FUNCTION_BLOCK FB_Power_lever
VAR_INPUT
	Forward:BOOL; (*Lever notch 1 forward*)
	Reverse:BOOL; (*Lever notch 1 reverse*)
	Pot:INT; (*Analogue value from lever potentiometer*)
	Button:BOOL;
	Neutral:BOOL; 
	Use_neutral:BOOL;
	Fully_fwd_val:INT; (*Value of analogue input when lever is fully forward*)
	Fully_rev_val:INT; (*Value of analogue input when lever is fully reverse*)
	Zero_deadband:INT; (*Lever zero position deadband on a scale of 0 to 10 000 i.e. a value of 100 gives a 1% deadband in each direction*)
	Full_lever_deadband:INT; (*Lever fully forward or reverse deadband on a scale of 0 to 10 000 i.e. a value of 100 gives a 1% deadband*)
	Notch_position:INT; (*Lever value (-10 000 to 10 000, no deadbands) at which forward and reverse notches change state*)
	Allowed_notch_variation:INT; (*Allowed variation in notch position*)
	Pos_out_of_range_val:INT; (*If the analogue Pot value exceeds this threshold, a fault will be generated.*)
	Neg_out_of_range_val:INT; (*If the analogue Pot value is less than this threshold, a fault will be generated.*)
END_VAR
VAR_OUTPUT
	Power_lever_data:dut_Power_lever;
	Raw:INT; (*Linear scaled lever value with no deadbands applied. -10 000 = fully reverse. +10 000 = fully forward.*)
	Linear:INT; (*Linear scaled lever value with deadbands applied. -10 000 = fully reverse. +10 000 = fully forward.*)
	Cubic:INT; (*Cubic scaling applied to lever value with deadbands applied. -10 000 = fully reverse. +10 000 = fully forward.*)
	cs_Forward_and_reverse:BOOL; (*Forward and reverse inputs both energised.*)
	cs_Pot_fwd_no_notch:BOOL; (*Pot shows that lever is forward but the forward notch is not activated*)
	cs_Pot_rev_no_notch:BOOL; (*Pot shows that lever is reverse but the reverse notch is not activated*)
	cs_Fwd_notch_not_pot:BOOL; (*Reverse notch is activated but the pot does not show that the lever is past the reverse notch*)
	cs_Rev_notch_not_pot:BOOL; (*Forward notch is activated but the pot does not show that the lever is past the forward notch*)
	cs_Out_of_range_pos:BOOL; (*The Pot value is out of range in the positive direction*)
	cs_Out_of_range_neg:BOOL; (*The Pot value is out of range in the negative direction*)
	hmi_data:dut_hmi_Power_lever; (*HMI status bits as well as Raw, Linear and Cubic values*)
END_VAR
VAR
	Linear_abs: INT;
	hmi_Word:WORD;
	TON_0: TON;
	TON_2: TON;
	TON_1: TON;
	TON_3: TON;
	Lever_scaling: Lever_scaling;
	Power_lever_data_m: Power_lever_data;
	Power_lever_faults: Power_lever_faults;
	BIT_TO_WORD_V0_0: FB_BIT_TO_WORD_V0;
END_VAR

Lever_scaling();
Power_lever_data_m();
Power_lever_faults();

METHOD Lever_scaling
VAR_INPUT
END_VAR
VAR_INST // added by the converter: edge detectors and wires of the graphical bodies
    _w1, _w2, _w3, _w4, _w5, _w6, _w8 : ANY;
    _w7 : REAL;
END_VAR
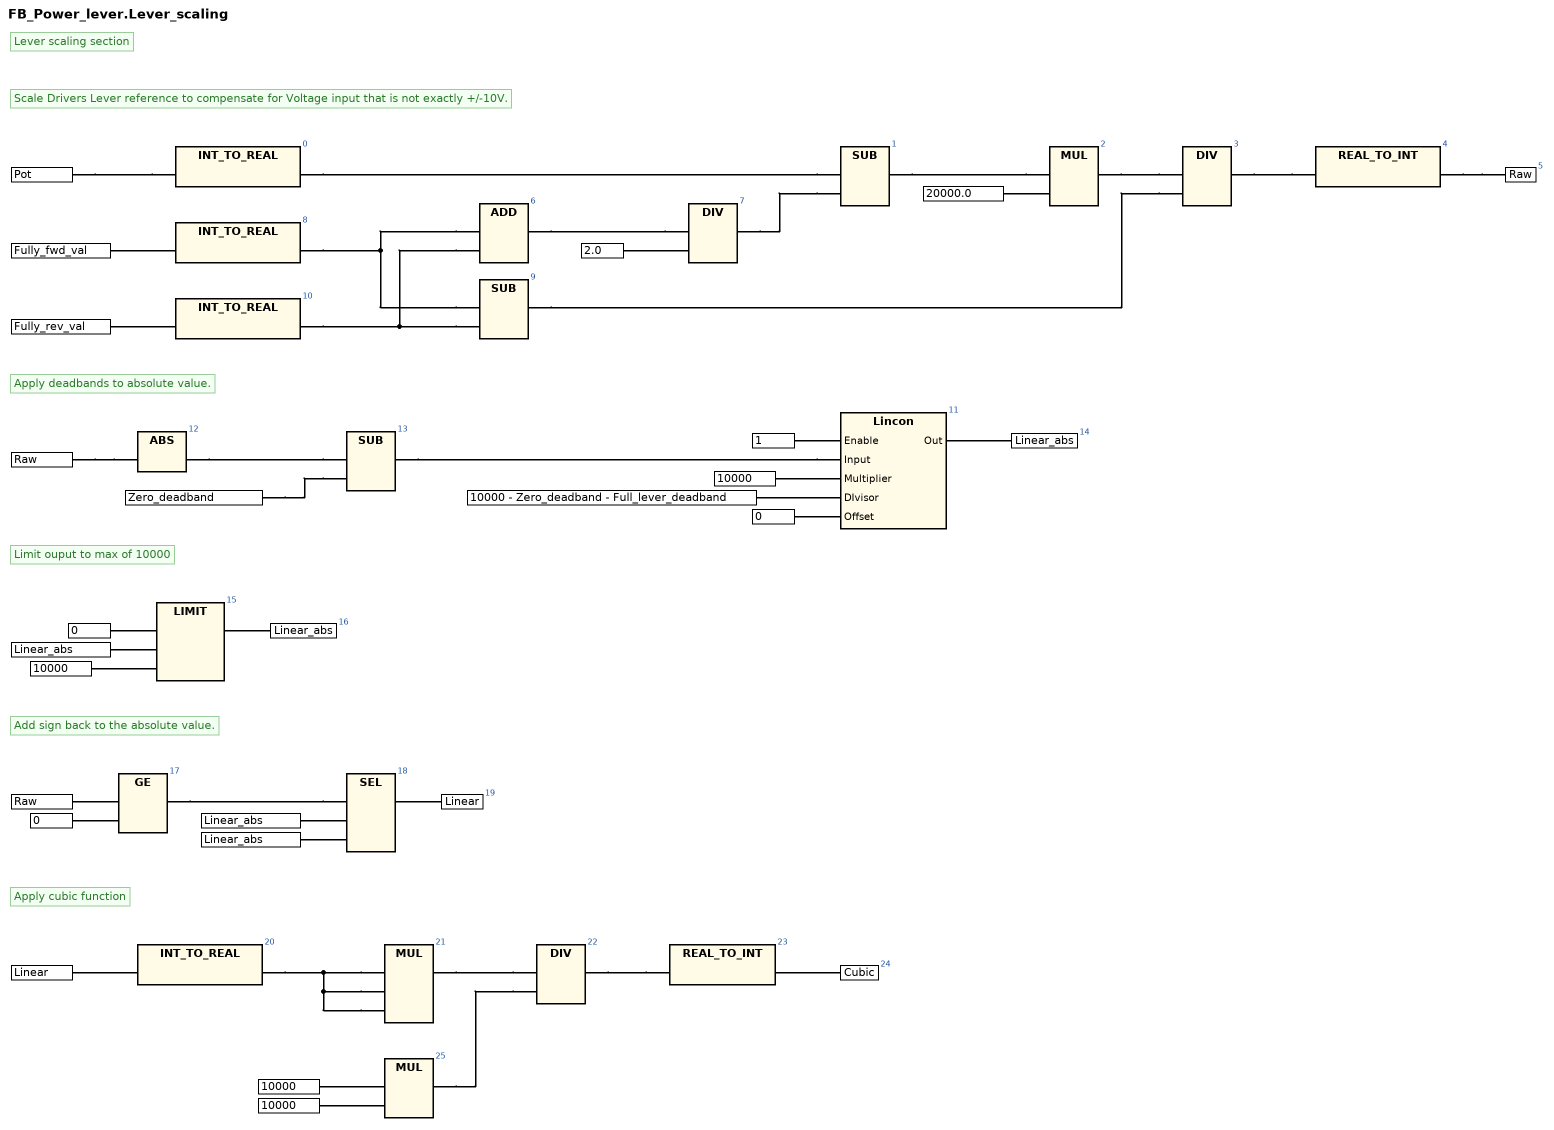
// Lever scaling section
// Scale Drivers Lever reference to compensate for Voltage input that is not exactly +/-10V.
Raw := REAL_TO_INT(((INT_TO_REAL(Pot) - _w1) * 20000.0) / _w2);
_w1 := (_w3 + _w4) / 2.0;
_w3 := INT_TO_REAL(Fully_fwd_val);
_w2 := _w3 - _w4;
_w4 := INT_TO_REAL(Fully_rev_val);
_w6 := Lincon(Enable := 1, Input := _w5, Multiplier := 10000, DIvisor := 10000 - Zero_deadband - Full_lever_deadband, Offset := 0);
// Apply deadbands to absolute value.
_w5 := ABS(Raw) - Zero_deadband;
Linear_abs := _w6;
// Limit ouput to max of 10000
Linear_abs := LIMIT(0, Linear_abs, 10000);
// Add sign back to the absolute value.
Linear := SEL(Raw >= 0, Linear_abs, Linear_abs);
// Apply cubic function
_w7 := INT_TO_REAL(Linear);
Cubic := REAL_TO_INT((_w7 * _w7 * _w7) / _w8);
_w8 := 10000 * 10000;
END_METHOD

METHOD Power_lever_data
VAR_INPUT
END_VAR

VAR
END_VAR
VAR_INST // added by the converter: edge detectors and wires of the graphical bodies
    _w1, _w3 : ANY;
    _w2, _w4, _w5 : BOOL;
END_VAR
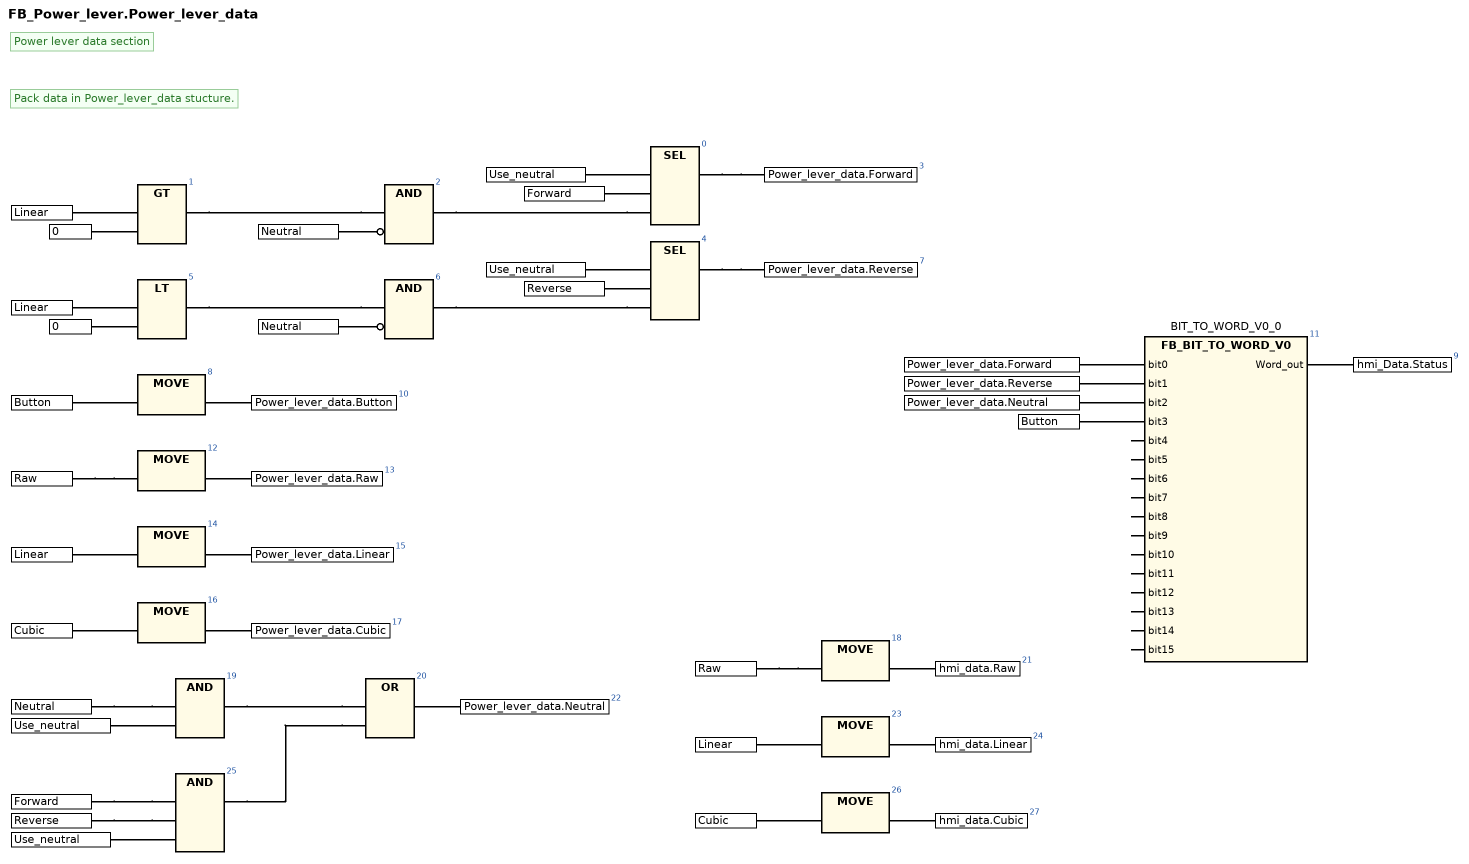
_w2 := SEL(Use_neutral, Forward, _w1);
// Power lever data section
// Pack data in Power_lever_data stucture.
_w1 := Linear > 0 AND NOT Neutral;
Power_lever_data.Forward := _w2;
_w4 := SEL(Use_neutral, Reverse, _w3);
_w3 := Linear < 0 AND NOT Neutral;
Power_lever_data.Reverse := _w4;
hmi_Data.Status := BIT_TO_WORD_V0_0.Word_out;
Power_lever_data.Button := Button;
BIT_TO_WORD_V0_0(
    bit0 := Power_lever_data.Forward,
    bit1 := Power_lever_data.Reverse,
    bit2 := Power_lever_data.Neutral,
    bit3 := Button); // FB_BIT_TO_WORD_V0
Power_lever_data.Raw := Raw;
Power_lever_data.Linear := Linear;
Power_lever_data.Cubic := Cubic;
hmi_data.Raw := Raw;
Power_lever_data.Neutral := Neutral AND Use_neutral OR _w5;
hmi_data.Linear := Linear;
_w5 := Forward AND Reverse AND Use_neutral;
hmi_data.Cubic := Cubic;
END_METHOD

METHOD Power_lever_faults
VAR_INPUT
END_VAR
VAR_INST // added by the converter: edge detectors and wires of the graphical bodies
    _w1, _w2, _w3, _w4 : ANY;
END_VAR
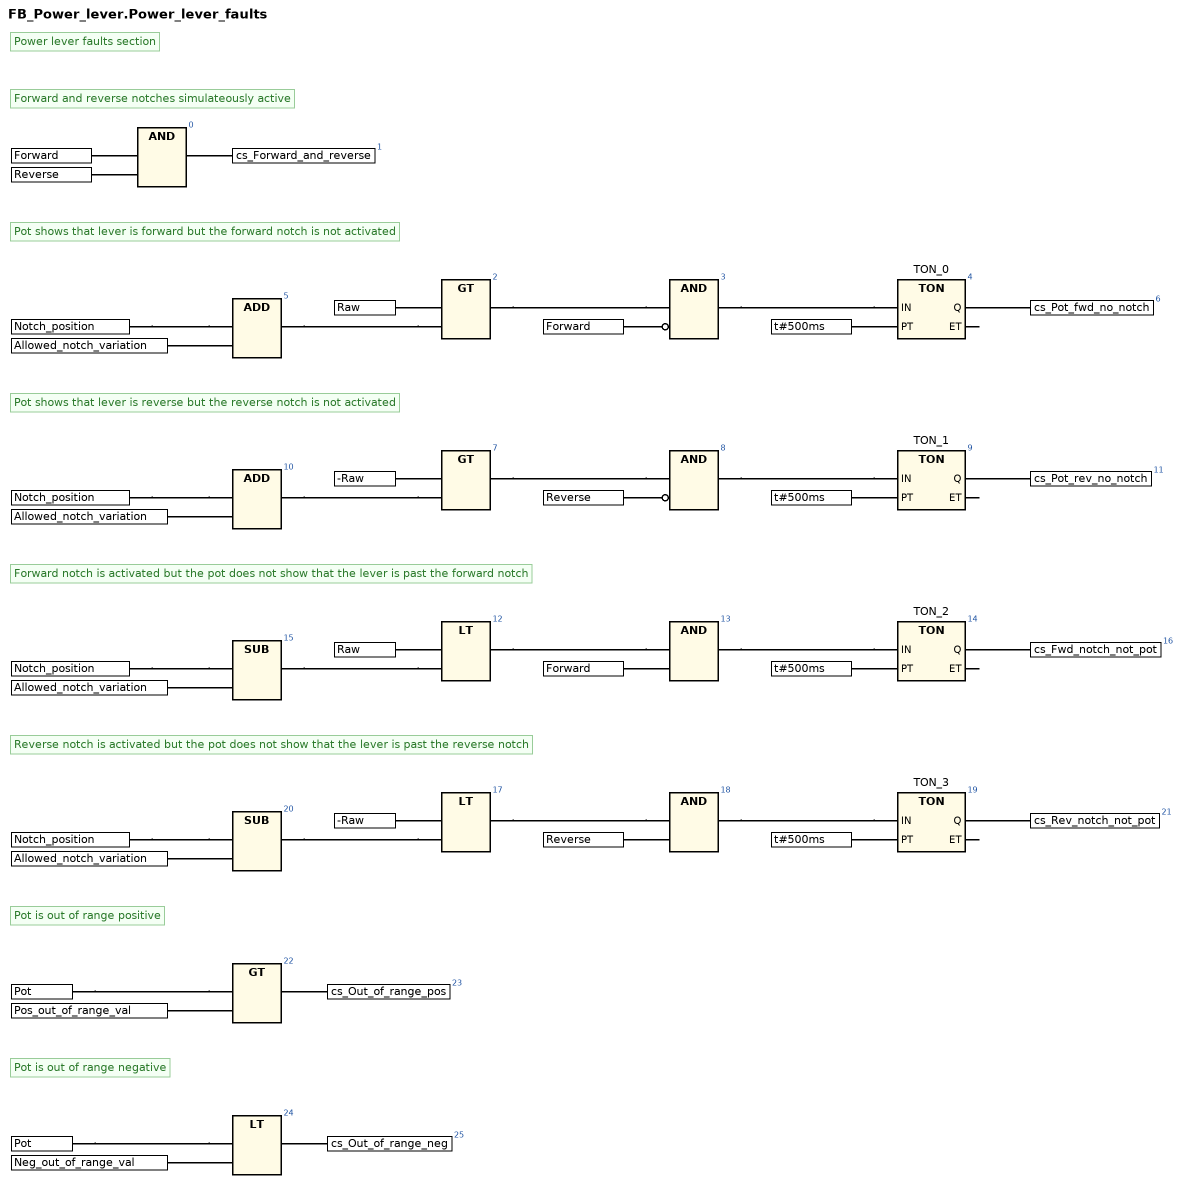
// Power lever faults section
// Forward and reverse notches simulateously active
cs_Forward_and_reverse := Forward AND Reverse;
TON_0(IN := Raw > _w1 AND NOT Forward, PT := t#500ms); // TON
// Pot shows that lever is forward but the forward notch is not activated
_w1 := Notch_position + Allowed_notch_variation;
cs_Pot_fwd_no_notch := TON_0.Q;
TON_1(IN := (-Raw) > _w2 AND NOT Reverse, PT := t#500ms); // TON
// Pot shows that lever is reverse but the reverse notch is not activated
_w2 := Notch_position + Allowed_notch_variation;
cs_Pot_rev_no_notch := TON_1.Q;
TON_2(IN := Raw < _w3 AND Forward, PT := t#500ms); // TON
// Forward notch is activated but the pot does not show that the lever is past the forward notch
_w3 := Notch_position - Allowed_notch_variation;
cs_Fwd_notch_not_pot := TON_2.Q;
TON_3(IN := (-Raw) < _w4 AND Reverse, PT := t#500ms); // TON
// Reverse notch is activated but the pot does not show that the lever is past the reverse notch
_w4 := Notch_position - Allowed_notch_variation;
cs_Rev_notch_not_pot := TON_3.Q;
// Pot is out of range positive
cs_Out_of_range_pos := Pot > Pos_out_of_range_val;
// Pot is out of range negative
cs_Out_of_range_neg := Pot < Neg_out_of_range_val;
END_METHOD

END_FUNCTION_BLOCK

(* stored: Version 1.1.0.1, ProductVersion 3.1.4024.0
   POU FB_Power_lever: Id {046c8a01-a8a9-4534-a6e7-75fa9037e7a8}, SpecialFunc None
   Method Lever_scaling: Id {7b5ae0f4-3ab8-4d60-a68c-cffda2f7d209}
   Method Power_lever_data: Id {967c78ca-ff9a-4630-99a4-ac6e2e7324eb}
   Method Power_lever_faults: Id {10b280ec-e8fd-4e5f-a3ae-353067d20ce1} *)
